INTERFACE I_EtherCatDiagnosticEventProvider EXTENDS I_EventReactionTcEvents

METHOD RaiseEtherCatDiagnosticEvent
VAR_INPUT
	EventId	  : UDINT;
	Argument1 : STRING := '';
	Argument2 : STRING := '';
	Argument3 : STRING := '';
END_VAR
END_METHOD

METHOD RaiseSyncUnitEvent
VAR_INPUT
	EventId	  : UDINT;
	Argument1 : STRING := '';
	Argument2 : STRING := '';
	Argument3 : STRING := '';
END_VAR
END_METHOD

END_INTERFACE

(* stored: Version 1.1.0.1, ProductVersion 3.1.4026.18
   Itf I_EtherCatDiagnosticEventProvider: Id {2b46d3ce-4575-4f3d-821d-77693f46da70}
   Method RaiseEtherCatDiagnosticEvent: Id {5bf6003a-71d5-43fb-912e-43a87a1d270b}
   Method RaiseSyncUnitEvent: Id {85e2b692-6448-4be0-b90d-317d7ce9edea} *)
